FUNCTION_BLOCK FB_PumpControl (* Basic Function Block Type *)
  (* Standard: 61499-2 *)
  (* Version 0.0, 2014-5-4, wildai, nxtControl GmbH, Template *)
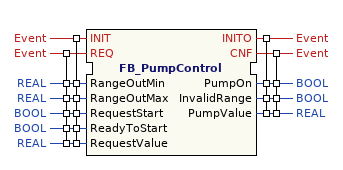
  EVENT_INPUT
    INIT WITH RangeOutMin, RangeOutMax, RequestStart, ReadyToStart, RequestValue; (* Initialization Request *)
    REQ WITH RangeOutMin, RangeOutMax, RequestStart, ReadyToStart, RequestValue; (* Normal Execution Request *)
  END_EVENT
  EVENT_OUTPUT
    INITO WITH PumpOn, InvalidRange, PumpValue; (* Initialization Confirm *)
    CNF WITH PumpOn, InvalidRange, PumpValue; (* Execution Confirmation *)
  END_EVENT
  VAR_INPUT
    RangeOutMin : REAL;
    RangeOutMax : REAL;
    RequestStart : BOOL;
    ReadyToStart : BOOL;
    RequestValue : REAL;
  END_VAR
  VAR_OUTPUT
    PumpOn : BOOL; (* Output event qualifier *)
    InvalidRange : BOOL;
    PumpValue : REAL;
  END_VAR
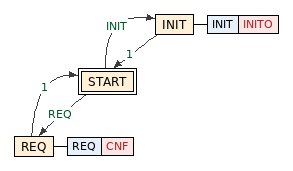
  EC_STATES
    START; (* Initial State *)
    INIT : INIT -> INITO; (* Initialization *)
    REQ : REQ -> CNF; (* Normal execution *)
  END_STATES
  EC_TRANSITIONS
    START TO INIT := INIT;
    INIT TO START := 1;
    START TO REQ := REQ;
    REQ TO START := 1;
  END_TRANSITIONS
  ALGORITHM INIT IN ST: (* Initialization algorithm *)
;

PumpOn := FALSE;
InvalidRange := FALSE;
PumpValue := 0.0;
  END_ALGORITHM
  ALGORITHM REQ IN ST: (* Normally executed algorithm *)
;

IF RequestStart AND ReadyToStart THEN
	IF RequestValue >= RangeOutMin AND RequestValue <= RangeOutMax THEN
		PumpValue := RequestValue;
		InvalidRange := FALSE;
		PumpOn := TRUE;
	ELSE
		PumpValue := 0.0;
		InvalidRange := TRUE;
		PumpOn := FALSE;
	END_IF;
ELSE
	PumpOn := FALSE;
	PumpValue := 0.0;
END_IF;
  END_ALGORITHM
END_FUNCTION_BLOCK
